{attribute 'GeneratedUsingTerminal: EP2339-0042-0017'}
{attribute addProperty BoxType "EP2339-0042-0017"}
{attribute addProperty Id "EtcSlaveTerminalBaseDI_X01_Pin4AT %I*DI_X01_Pin_830843C11DI_X01_Pin2AT %I*DI_X01_Pin_830843C11DI_X02_Pin4AT %I*DI_X02_Pin_830843C11DI_X02_Pin2AT %I*DI_X02_Pin_830843C11DI_X03_Pin4AT %I*DI_X03_Pin_830843C11DI_X03_Pin2AT %I*DI_X03_Pin_830843C11DI_X04_Pin4AT %I*DI_X04_Pin_830843C11DI_X04_Pin2AT %I*DI_X04_Pin_830843C11DI_X05_Pin4AT %I*DI_X05_Pin_830843C11DI_X05_Pin2AT %I*DI_X05_Pin_830843C11DI_X06_Pin4AT %I*DI_X06_Pin_830843C11DI_X06_Pin2AT %I*DI_X06_Pin_830843C11DI_X07_Pin4AT %I*DI_X07_Pin_830843C11DI_X07_Pin2AT %I*DI_X07_Pin_830843C11DI_X08_Pin4AT %I*DI_X08_Pin_830843C11DI_X08_Pin2AT %I*DI_X08_Pin_830843C11DO_X01_Pin_4AT %Q*DO_X01_Pin_42CA91F71DO_X01_Pin_2AT %Q*DO_X01_Pin_42CA91F71DO_X02_Pin_4AT %Q*DO_X02_Pin_42CA91F71DO_X02_Pin_2AT %Q*DO_X02_Pin_42CA91F71DO_X03_Pin_4AT %Q*DO_X03_Pin_42CA91F71DO_X03_Pin_2AT %Q*DO_X03_Pin_42CA91F71DO_X04_Pin_4AT %Q*DO_X04_Pin_42CA91F71DO_X04_Pin_2AT %Q*DO_X04_Pin_42CA91F71DO_X05_Pin_4AT %Q*DO_X05_Pin_42CA91F71DO_X05_Pin_2AT %Q*DO_X05_Pin_42CA91F71DO_X06_Pin_4AT %Q*DO_X06_Pin_42CA91F71DO_X06_Pin_2AT %Q*DO_X06_Pin_42CA91F71DO_X07_Pin_4AT %Q*DO_X07_Pin_42CA91F71DO_X07_Pin_2AT %Q*DO_X07_Pin_42CA91F71DO_X08_Pin_4AT %Q*DO_X08_Pin_42CA91F71DO_X08_Pin_2AT %Q*DO_X08_Pin_42CA91F71WcStateAT %I*WcState_9091E0EB2InfoDataAT %I*InfoData_6F19DB2B2"}
{attribute addProperty CRC "98535135"}
{attribute addProperty Size "36"}
TYPE EP2339_05DF86DF EXTENDS EtcSlaveTerminalBase :
STRUCT
	{attribute addProperty Name "DI_X01_Pin4"}
	DI_X01_Pin4 : DI_X01_Pin_830843C1;
	{attribute addProperty Name "DI_X01_Pin2"}
	DI_X01_Pin2 : DI_X01_Pin_830843C1;
	{attribute addProperty Name "DI_X02_Pin4"}
	DI_X02_Pin4 : DI_X02_Pin_830843C1;
	{attribute addProperty Name "DI_X02_Pin2"}
	DI_X02_Pin2 : DI_X02_Pin_830843C1;
	{attribute addProperty Name "DI_X03_Pin4"}
	DI_X03_Pin4 : DI_X03_Pin_830843C1;
	{attribute addProperty Name "DI_X03_Pin2"}
	DI_X03_Pin2 : DI_X03_Pin_830843C1;
	{attribute addProperty Name "DI_X04_Pin4"}
	DI_X04_Pin4 : DI_X04_Pin_830843C1;
	{attribute addProperty Name "DI_X04_Pin2"}
	DI_X04_Pin2 : DI_X04_Pin_830843C1;
	{attribute addProperty Name "DI_X05_Pin4"}
	DI_X05_Pin4 : DI_X05_Pin_830843C1;
	{attribute addProperty Name "DI_X05_Pin2"}
	DI_X05_Pin2 : DI_X05_Pin_830843C1;
	{attribute addProperty Name "DI_X06_Pin4"}
	DI_X06_Pin4 : DI_X06_Pin_830843C1;
	{attribute addProperty Name "DI_X06_Pin2"}
	DI_X06_Pin2 : DI_X06_Pin_830843C1;
	{attribute addProperty Name "DI_X07_Pin4"}
	DI_X07_Pin4 : DI_X07_Pin_830843C1;
	{attribute addProperty Name "DI_X07_Pin2"}
	DI_X07_Pin2 : DI_X07_Pin_830843C1;
	{attribute addProperty Name "DI_X08_Pin4"}
	DI_X08_Pin4 : DI_X08_Pin_830843C1;
	{attribute addProperty Name "DI_X08_Pin2"}
	DI_X08_Pin2 : DI_X08_Pin_830843C1;
	{attribute addProperty Name "DO_X01_Pin_4"}
	DO_X01_Pin_4 : DO_X01_Pin_42CA91F7;
	{attribute addProperty Name "DO_X01_Pin_2"}
	DO_X01_Pin_2 : DO_X01_Pin_42CA91F7;
	{attribute addProperty Name "DO_X02_Pin_4"}
	DO_X02_Pin_4 : DO_X02_Pin_42CA91F7;
	{attribute addProperty Name "DO_X02_Pin_2"}
	DO_X02_Pin_2 : DO_X02_Pin_42CA91F7;
	{attribute addProperty Name "DO_X03_Pin_4"}
	DO_X03_Pin_4 : DO_X03_Pin_42CA91F7;
	{attribute addProperty Name "DO_X03_Pin_2"}
	DO_X03_Pin_2 : DO_X03_Pin_42CA91F7;
	{attribute addProperty Name "DO_X04_Pin_4"}
	DO_X04_Pin_4 : DO_X04_Pin_42CA91F7;
	{attribute addProperty Name "DO_X04_Pin_2"}
	DO_X04_Pin_2 : DO_X04_Pin_42CA91F7;
	{attribute addProperty Name "DO_X05_Pin_4"}
	DO_X05_Pin_4 : DO_X05_Pin_42CA91F7;
	{attribute addProperty Name "DO_X05_Pin_2"}
	DO_X05_Pin_2 : DO_X05_Pin_42CA91F7;
	{attribute addProperty Name "DO_X06_Pin_4"}
	DO_X06_Pin_4 : DO_X06_Pin_42CA91F7;
	{attribute addProperty Name "DO_X06_Pin_2"}
	DO_X06_Pin_2 : DO_X06_Pin_42CA91F7;
	{attribute addProperty Name "DO_X07_Pin_4"}
	DO_X07_Pin_4 : DO_X07_Pin_42CA91F7;
	{attribute addProperty Name "DO_X07_Pin_2"}
	DO_X07_Pin_2 : DO_X07_Pin_42CA91F7;
	{attribute addProperty Name "DO_X08_Pin_4"}
	DO_X08_Pin_4 : DO_X08_Pin_42CA91F7;
	{attribute addProperty Name "DO_X08_Pin_2"}
	DO_X08_Pin_2 : DO_X08_Pin_42CA91F7;
	{attribute addProperty Name "WcState"}
	WcState : WcState_9091E0EB;
	{attribute addProperty Name "InfoData"}
	InfoData : InfoData_6F19DB2B;
END_STRUCT
END_TYPE

(* stored: Version 1.2.0.0, ProductVersion 3.1.4024.9
   DUT EP2339_05DF86DF: Id {02edb030-3733-44e7-8630-8887d3790e6c} *)
